// TIA Portal V17 export
// export: Created 2025-06-26T06:49:14.7827418Z, ExportSetting WithDefaults, DisplayName Totally Integrated Automation Portal, DisplayVersion V17 Update 8, DisplayName TIA Portal Openness, DisplayVersion V17 Update 8, DisplayName TIA Portal Version Control Interface, DisplayVersion V17, DisplayName STEP 7 Professional, DisplayVersion V17 Update 8, DisplayName STEP 7 Safety, DisplayVersion V17 Update 6, DisplayName WinCC Advanced, DisplayVersion V17 Update 8
FUNCTION_BLOCK "ApplicationCommunication"   // FB6, LAD
{ S7_Optimized_Access := 'TRUE' }
VERSION : 0.1
// Note some networks are in Ladder because the FBD equivalents are too bulky and the SCL equivalents are too easy to screw up accidentally.
// stored: AutoNumber true, IsIECCheckEnabled false, IsRetainMemResEnabled false, MemoryReserve 0, SetENOAutomatically false, UDAEnableTagReadback false
   VAR
      ExpansionRegulatorManualOn { ExternalAccessible := 'False'; ExternalVisible := 'False'; ExternalWritable := 'False'} : Bool;
      ExpansionRegulatorManualOff { ExternalAccessible := 'False'; ExternalVisible := 'False'; ExternalWritable := 'False'; S7_SetPoint := 'True'} : Bool;
      HeatSinkOutManualOn { ExternalAccessible := 'False'; ExternalVisible := 'False'; ExternalWritable := 'False'} : Bool;
      HeatSinkOutManualOff { ExternalAccessible := 'False'; ExternalVisible := 'False'; ExternalWritable := 'False'} : Bool;
      PerformanceManualModeOn { ExternalAccessible := 'False'; ExternalVisible := 'False'; ExternalWritable := 'False'} : Bool;
      PerformanceManualModeOff { ExternalAccessible := 'False'; ExternalVisible := 'False'; ExternalWritable := 'False'} : Bool;
      OilHeatingManualOn { ExternalAccessible := 'False'; ExternalVisible := 'False'; ExternalWritable := 'False'} : Bool;
      OilHeatingManualOff { ExternalAccessible := 'False'; ExternalVisible := 'False'; ExternalWritable := 'False'} : Bool;
      PinchManualModeOn { ExternalAccessible := 'False'; ExternalVisible := 'False'; ExternalWritable := 'False'} : Bool;
      PinchManualModeOff { ExternalAccessible := 'False'; ExternalVisible := 'False'; ExternalWritable := 'False'} : Bool;
      SuperheatManualOn { ExternalAccessible := 'False'; ExternalVisible := 'False'; ExternalWritable := 'False'} : Bool;
      SuperheatManualOff { ExternalAccessible := 'False'; ExternalVisible := 'False'; ExternalWritable := 'False'} : Bool;
      AlarmAckOn { ExternalAccessible := 'False'; ExternalVisible := 'False'; ExternalWritable := 'False'} : Bool;
      AlarmAckOff { ExternalAccessible := 'False'; ExternalVisible := 'False'; ExternalWritable := 'False'} : Bool;
      ResetEstopOn { ExternalAccessible := 'False'; ExternalVisible := 'False'; ExternalWritable := 'False'} : Bool;
      ResetEstopOff { ExternalAccessible := 'False'; ExternalVisible := 'False'; ExternalWritable := 'False'} : Bool;
      FastStopOn { ExternalAccessible := 'False'; ExternalVisible := 'False'; ExternalWritable := 'False'} : Bool;
      ExpansionManualPrev { ExternalAccessible := 'False'; ExternalVisible := 'False'; ExternalWritable := 'False'} : Real;
      HeatSinkManualPrev { ExternalAccessible := 'False'; ExternalVisible := 'False'; ExternalWritable := 'False'} : Real;
      PerformanceManualPrev { ExternalAccessible := 'False'; ExternalVisible := 'False'; ExternalWritable := 'False'} : Real;
      OilHeatingManualPrev { ExternalAccessible := 'False'; ExternalVisible := 'False'; ExternalWritable := 'False'} : Real;
      PinchManualPrev { ExternalAccessible := 'False'; ExternalVisible := 'False'; ExternalWritable := 'False'} : Real;
      SuperheatManualPrev { ExternalAccessible := 'False'; ExternalVisible := 'False'; ExternalWritable := 'False'} : Real;
      HeatboosterSetpointPrev { ExternalAccessible := 'False'; ExternalVisible := 'False'; ExternalWritable := 'False'} : Real;
      RegulationTargetPrev { ExternalAccessible := 'False'; ExternalVisible := 'False'; ExternalWritable := 'False'} : Int;
      S7Watchdog : "fbHeartbeatCount2";
   END_VAR
   VAR_TEMP
      bDummy : Bool;
      fDummy : Real;
   END_VAR
   VAR_TEMP   // added for the SCL form of the ladder/FBD networks
      _w1 : Bool;
      _w2 : Bool;
      _w3 : Bool;
      _w4 : Bool;
      _w5 : Bool;
      _w6 : Bool;
      _w7 : Bool;
      _w8 : Bool;
      _w9 : Bool;
      _w10 : Bool;
   END_VAR
BEGIN

REGION Network 1 (SCL): Status
   // Applications PLC GETs these.
   "DB_Application".FromHB.EmergencyStop       := "DB_System".bEmergencyStop;
   "DB_Application".FromHB.OilHeatersGroup1    := "DB_DO".HBL_EC_01;
   "DB_Application".FromHB.OilHeatersGroup2    := "DB_DO".HBL_EC_02;
   "DB_Application".FromHB.HBL_SC_10_Ready     := "DB_InverterDrives".HBL_SC_10.Stat.bReady;
   "DB_Application".FromHB.HBL_SC_10_Run       := "DB_InverterDrives".HBL_SC_10.Stat.bRun;
   "DB_Application".FromHB.HBL_HV_630           := "DB_DO".HBL_HV_630;
   "DB_Application".FromHB.CPC_P_01            := "DB_DO".CPC_P_01;
   "DB_Application".FromHB.SSC_P_01            := "DB_DO".SSC_P_01;
   "DB_Application".FromHB.HBL_SC_10_Tripped   := "DB_InverterDrives".HBL_SC_10.Stat.bTrip;
   "DB_Application".FromHB.HBL_SC_02_Ready     := "DB_InverterDrives".HBL_SC_02.Stat.bReady;
   "DB_Application".FromHB.HBL_SC_02_Run       := "DB_InverterDrives".HBL_SC_02.Stat.bRun;
   "DB_Application".FromHB.HBL_SC_02_Tripped   := "DB_InverterDrives".HBL_SC_02.Stat.bTrip;
   "DB_Application".FromHB.SSC_F_01            := "DB_DO".SSC_F_01;
   "DB_Application".FromHB.SSC_P_02            := "DB_DO".SSC_P_02;
   "DB_Application".FromHB.HBL_LS_01           := "DB_DI".HBL_LS_01.bValue;
   "DB_Application".FromHB.HBL_LS_02           := "DB_DI".HBL_LS_02.bValue;
   "DB_Application".FromHB.MachineState        := "DB_State".State.State_Number;
   "DB_Application".FromHB.CompressorType      := "DB_CurrentSetting".Compressor.CompressorTypeNumber;
   "DB_Application".FromHB.SystemType          := "DB_CurrentSetting".System.SystemTypeNumber;
   "DB_Application".FromHB.RefrigerantType     := "DB_CurrentSetting".Fluid.FluidTypeNumber;
   "DB_Application".FromHB.UptimeHours         := UDINT_TO_INT("DB_System".SystemUptime.nHours);
   "DB_Application".FromHB.UptimeMinutes       := "DB_System".SystemUptime.nMinutes;
   "DB_Application".FromHB.UptimeSeconds       := "DB_System".SystemUptime.nSeconds;
   "DB_Application".FromHB.ActiveTimeHours     := UDINT_TO_INT("DB_System".SystemActiveTime.nHours);
   "DB_Application".FromHB.ActiveTimeMinutes   := "DB_System".SystemActiveTime.nMinutes;
   "DB_Application".FromHB.ActiveTimeSeconds   := "DB_System".SystemActiveTime.nSeconds;
   "DB_Application".FromHB.RunningTimeHours    := UDINT_TO_INT("DB_System".RunningTime.nHours);
   "DB_Application".FromHB.RunningTimeMinutes  := "DB_System".RunningTime.nMinutes;
   "DB_Application".FromHB.RunningTimeSeconds  := "DB_System".RunningTime.nSeconds;
   "DB_Application".FromHB.HeatboosterSetpoint := "DB_Regulators".HeatboosterSetpoint;
   "DB_Application".FromHB.RegulationTarget    := "DB_Regulators".RegulationTarget;
   "DB_Application".FromHB.HBL_HCV_514_Force   := FALSE; // ###FIX
   "DB_Application".FromHB.HBL_HCV_514         := 5.14; //##FIX
   "DB_Application".FromHB.HBL_HCV_548_Force   := FALSE; // ##FIX
   "DB_Application".FromHB.HBL_HCV_548         := 5.48; //##FIX
END_REGION

REGION Network 2 (SCL): DB_AI
   // Copy only .fValues for minimum bandwidth
   "DB_Application".FromHB.DB_AI.HBL_TT_502 := "DB_AI".HBL_TT_502.Eng.fValue;
   "DB_Application".FromHB.DB_AI.HBL_PT_503 := "DB_AI".HBL_PT_503.Eng.fValue;
   "DB_Application".FromHB.DB_AI.HBL_TT_504 := "DB_AI".HBL_TT_504.Eng.fValue;
   "DB_Application".FromHB.DB_AI.HBL_LT_510 := "DB_AI".HBL_LT_510.Eng.fValue;
   "DB_Application".FromHB.DB_AI.HBL_PT_511 := "DB_AI".HBL_PT_511.Eng.fValue;
   "DB_Application".FromHB.DB_AI.HBL_TT_512 := "DB_AI".HBL_TT_512.Eng.fValue;
   "DB_Application".FromHB.DB_AI.HBL_TT_516 := "DB_AI".HBL_TT_516.Eng.fValue;
   "DB_Application".FromHB.DB_AI.HBL_PT_517 := "DB_AI".HBL_PT_517.Eng.fValue;
   "DB_Application".FromHB.DB_AI.HBL_TT_518 := "DB_AI".HBL_TT_518.Eng.fValue;
   "DB_Application".FromHB.DB_AI.HBL_PT_519 := "DB_AI".HBL_PT_519.Eng.fValue;
   "DB_Application".FromHB.DB_AI.HBL_FT_520 := "DB_AI".HBL_FT_520.Eng.fValue;
   "DB_Application".FromHB.DB_AI.HBL_TT_530 := "DB_AI".HBL_TT_530.Eng.fValue;
   "DB_Application".FromHB.DB_AI.HBL_PT_531 := "DB_AI".HBL_PT_531.Eng.fValue;
   "DB_Application".FromHB.DB_AI.HBL_TT_532 := "DB_AI".HBL_TT_532.Eng.fValue;
   "DB_Application".FromHB.DB_AI.HBL_TT_533 := "DB_AI".HBL_TT_533.Eng.fValue;
   "DB_Application".FromHB.DB_AI.HBL_PT_534 := "DB_AI".HBL_PT_534.Eng.fValue;
   "DB_Application".FromHB.DB_AI.HBL_AT_535 := "DB_AI".HBL_AT_535.Eng.fValue;
   "DB_Application".FromHB.DB_AI.HBL_TT_540 := "DB_AI".HBL_TT_540.Eng.fValue;
   "DB_Application".FromHB.DB_AI.HBL_PT_541 := "DB_AI".HBL_PT_541.Eng.fValue;
   "DB_Application".FromHB.DB_AI.HBL_TT_542 := "DB_AI".HBL_TT_542.Eng.fValue;
   "DB_Application".FromHB.DB_AI.HBL_TT_543 := "DB_AI".HBL_TT_543.Eng.fValue;
   "DB_Application".FromHB.DB_AI.HBL_PT_544 := "DB_AI".HBL_PT_544.Eng.fValue;
   "DB_Application".FromHB.DB_AI.HBL_AT_545 := "DB_AI".HBL_AT_545.Eng.fValue;
   "DB_Application".FromHB.DB_AI.HBL_TT_546 := "DB_AI".HBL_TT_546.Eng.fValue;
   "DB_Application".FromHB.DB_AI.HBL_PT_547 := "DB_AI".HBL_PT_547.Eng.fValue;
   "DB_Application".FromHB.DB_AI.HBL_TT_571 := "DB_AI".HBL_TT_571.Eng.fValue;
   "DB_Application".FromHB.DB_AI.HBL_PT_572 := "DB_AI".HBL_PT_572.Eng.fValue;
   "DB_Application".FromHB.DB_AI.HBL_TT_573 := "DB_AI".HBL_TT_573.Eng.fValue;
   "DB_Application".FromHB.DB_AI.HBL_LT_610 := "DB_AI".HBL_LT_610.Eng.fValue;
   "DB_Application".FromHB.DB_AI.HBL_TT_611 := "DB_AI".HBL_TT_611.Eng.fValue;
   "DB_Application".FromHB.DB_AI.HBL_PT_612 := "DB_AI".HBL_PT_612.Eng.fValue;
   "DB_Application".FromHB.DB_AI.HBL_CT_615 := "DB_AI".HBL_CT_615.Eng.fValue;
   "DB_Application".FromHB.DB_AI.HBL_PT_618 := "DB_AI".HBL_PT_618.Eng.fValue;
   "DB_Application".FromHB.DB_AI.HBL_PT_635 := "DB_AI".HBL_PT_635.Eng.fValue;
   "DB_Application".FromHB.DB_AI.HBL_PT_636 := "DB_AI".HBL_PT_636.Eng.fValue;
   "DB_Application".FromHB.DB_AI.HBL_LT_650 := "DB_AI".HBL_LT_650.Eng.fValue;
   "DB_Application".FromHB.DB_AI.HBL_PT_651 := "DB_AI".HBL_PT_651.Eng.fValue;
   "DB_Application".FromHB.DB_AI.HBL_PT_701 := "DB_AI".HBL_PT_701.Eng.fValue;
   "DB_Application".FromHB.DB_AI.HBL_PT_702 := "DB_AI".HBL_PT_702.Eng.fValue;
   "DB_Application".FromHB.DB_AI.HBL_PT_703 := "DB_AI".HBL_PT_703.Eng.fValue;

   "DB_Application".FromHB.DB_AI.CPC_LT_870 := "DB_AI".CPC_LT_870.Eng.fValue;
   "DB_Application".FromHB.DB_AI.CPC_TT_871 := "DB_AI".CPC_TT_871.Eng.fValue;
   "DB_Application".FromHB.DB_AI.CPC_PT_872 := "DB_AI".CPC_PT_872.Eng.fValue;
   "DB_Application".FromHB.DB_AI.CPC_PT_862 := "DB_AI".CPC_PT_862.Eng.fValue;
   "DB_Application".FromHB.DB_AI.HBL_TT_901 := "DB_AI".HBL_TT_901.Eng.fValue;
   "DB_Application".FromHB.DB_AI.HBL_PT_902 := "DB_AI".HBL_PT_902.Eng.fValue;

   "DB_Application".FromHB.DB_AI.HBL_TT_03 := "DB_AI".HBL_TT_03.Eng.fValue;
   "DB_Application".FromHB.DB_AI.HBL_TT_16 := "DB_AI".HBL_TT_16.Eng.fValue;
   "DB_Application".FromHB.DB_AI.HBL_TT_17 := "DB_AI".HBL_TT_17.Eng.fValue;
   "DB_Application".FromHB.DB_AI.HBL_TT_18 := "DB_AI".HBL_TT_18.Eng.fValue;
   "DB_Application".FromHB.DB_AI.HBL_TT_20 := "DB_AI".HBL_TT_20.Eng.fValue;
   "DB_Application".FromHB.DB_AI.HBL_TT_21 := "DB_AI".HBL_TT_21.Eng.fValue;
   "DB_Application".FromHB.DB_AI.HBL_TT_22 := "DB_AI".HBL_TT_22.Eng.fValue;
   "DB_Application".FromHB.DB_AI.HBL_TT_23 := "DB_AI".HBL_TT_23.Eng.fValue;
   "DB_Application".FromHB.DB_AI.HBL_TT_24 := "DB_AI".HBL_TT_24.Eng.fValue;
   "DB_Application".FromHB.DB_AI.HBL_TT_25 := "DB_AI".HBL_TT_25.Eng.fValue;
   "DB_Application".FromHB.DB_AI.HBL_TT_26 := "DB_AI".HBL_TT_26.Eng.fValue;
   "DB_Application".FromHB.DB_AI.HBL_TT_27 := "DB_AI".HBL_TT_27.Eng.fValue;
   "DB_Application".FromHB.DB_AI.HBL_PT_05 := "DB_AI".HBL_PT_05.Eng.fValue;
   "DB_Application".FromHB.DB_AI.HBL_PT_06 := "DB_AI".HBL_PT_960.Eng.fValue;
   "DB_Application".FromHB.DB_AI.HBL_PT_17 := "DB_AI".HBL_PT_961.Eng.fValue;
   "DB_Application".FromHB.DB_AI.HBL_CT_01 := "DB_AI".HBL_CT_01.Eng.fValue;
   "DB_Application".FromHB.DB_AI.HBL_CT_03 := "DB_AI".HBL_CT_950.Eng.fValue;

   "DB_Application".FromHB.DB_AI.SSC_TT_01 := "DB_AI".SSC_TT_01.Eng.fValue;
   "DB_Application".FromHB.DB_AI.SSC_TT_02 := "DB_AI".SSC_TT_02.Eng.fValue;
   "DB_Application".FromHB.DB_AI.SSC_TT_03 := "DB_AI".SSC_TT_03.Eng.fValue;
   "DB_Application".FromHB.DB_AI.SSC_TT_04 := "DB_AI".SSC_TT_04.Eng.fValue;
   "DB_Application".FromHB.DB_AI.SSC_PIT_01 := "DB_AI".SSC_PIT_01.Eng.fValue;
   "DB_Application".FromHB.DB_AI.SSC_PDT_01 := "DB_AI".SSC_PDT_01.Eng.fValue;
   "DB_Application".FromHB.DB_AI.SSC_LT_01 := "DB_AI".SSC_LT_01.Eng.fValue;
END_REGION

REGION Network 3 (SCL): DB_Calc
   // Done this way for minimum bandwidth
   "DB_Application".FromHB.DB_Calc.Compressor_CrankcaseSaturationTemperature   := "DB_Calc".Compressor.CrankcaseSaturationTemperature.fValue;
   "DB_Application".FromHB.DB_Calc.Compressor_CrankcaseSuperheat               := "DB_Calc".Compressor.CrankcaseSuperheat.fValue;
   "DB_Application".FromHB.DB_Calc.Compressor_VolumetricEfficiency             := "DB_Calc".Compressor.VolumetricEfficiency.fValue;
   "DB_Application".FromHB.DB_Calc.Compressor_IsentropicEfficiency             := "DB_Calc".Compressor.IsentropicEfficiency.fValue;
   "DB_Application".FromHB.DB_Calc.Compressor_Massflow                         := "DB_Calc".Compressor.Massflow.fValue;

   "DB_Application".FromHB.DB_Calc.Heatsink_DeltaT                             := "DB_Calc".HeatSink.DeltaT.fValue;
   "DB_Application".FromHB.DB_Calc.Heatsink_Pinch                              := "DB_Calc".HeatSink.Pinch.fValue;
   "DB_Application".FromHB.DB_Calc.Heatsink_Heatrate                           := "DB_Calc".HeatSink.HeatRate.fValue;
   "DB_Application".FromHB.DB_Calc.Heatsink_DeltaP                             := "DB_Calc".HeatSink.DeltaP.fValue;
   "DB_Application".FromHB.DB_Calc.Heatsink_Massflow                           := "DB_Calc".HeatSink.Massflow.fValue;

   "DB_Application".FromHB.DB_Calc.Heatsource_DeltaT                           := "DB_Calc".HeatSource.DeltaT.fValue;
   "DB_Application".FromHB.DB_Calc.Heatsource_Pinch                            := "DB_Calc".HeatSource.Pinch.fValue;
   "DB_Application".FromHB.DB_Calc.Heatsource_Heatrate                         := "DB_Calc".HeatSource.HeatRate.fValue;
   "DB_Application".FromHB.DB_Calc.Heatsource_DeltaP                           := "DB_Calc".HeatSource.DeltaP.fValue;
   "DB_Application".FromHB.DB_Calc.Heatsource_Massflow                         := "DB_Calc".HeatSource.Massflow.fValue;
   "DB_Application".FromHB.DB_Calc.Heatsource_TemperatureRateOfChange          := "DB_Calc".HeatSource.TemperatureRateOfChange.fValue;

   "DB_Application".FromHB.DB_Calc.HighPressPart_CompressorSaturationTemperature := "DB_Calc".HighPressPart.CompressorSaturationTemperature.fValue;
   "DB_Application".FromHB.DB_Calc.HighPressPart_CompressorSuperheat           := "DB_Calc".HighPressPart.CompressorSuperheat.fValue;
   "DB_Application".FromHB.DB_Calc.HighPressPart_CondenserSaturationTemperature:= "DB_Calc".HighPressPart.CondenserSaturationTemperature.fValue;
   "DB_Application".FromHB.DB_Calc.HighPressPart_CondenserSubcooling           := "DB_Calc".HighPressPart.CondenserSubcooling.fValue;
   "DB_Application".FromHB.DB_Calc.HighPressPart_ExpansionValveSubcooling      := "DB_Calc".HighPressPart.ExpansionValveSubcooling.fValue;
   "DB_Application".FromHB.DB_Calc.HighPressPart_CondenserDeltaP               := "DB_Calc".HighPressPart.CondenserDeltaP.fValue;

   "DB_Application".FromHB.DB_Calc.LowPressPart_EvaporatorSuperheat            := "DB_Calc".LowPressPart.EvaporatorSuperheat.fValue;
   "DB_Application".FromHB.DB_Calc.LowPressPart_CompressorSuperheat            := "DB_Calc".LowPressPart.CompressorSuperheat.fValue;
   "DB_Application".FromHB.DB_Calc.LowPressPart_EvaporatorSaturationTemperature:= "DB_Calc".LowPressPart.EvaporatorSaturationTemperature.fValue;
   "DB_Application".FromHB.DB_Calc.LowPressPart_CompressorSaturationTemperature:= "DB_Calc".LowPressPart.CompressorSaturationTemperature.fValue;

   "DB_Application".FromHB.DB_Calc.System_Quality                              := "DB_Calc".System.Quality.fValue;
   "DB_Application".FromHB.DB_Calc.System_COP                                  := "DB_Calc".System.COP.fValue;
   "DB_Application".FromHB.DB_Calc.System_ElectricalPower                      := "DB_Calc".System.ElectricalPower.fValue;
   "DB_Application".FromHB.DB_Calc.System_TemperatureLift                      := "DB_Calc".System.TemperatureLift.fValue;
   "DB_Application".FromHB.DB_Calc.System_MotorEfficiency                      := "DB_Calc".System.MotorEfficiency.fValue;
   "DB_Application".FromHB.DB_Calc.System_FMEP                                 := "DB_Calc".System.FMEP.fValue;

   "DB_Application".FromHB.DB_Calc.Aux_ShaftSealDeltaT                         := "DB_Calc".Auxiliary.ShaftSealDeltaT.fValue;
   "DB_Application".FromHB.DB_Calc.Aux_CPCPumpDeltaP                           := "DB_Calc".Auxiliary.CPCDeltaP.fValue;

   "DB_Application".FromHB.DB_Calc.Misc_EvaporatorDischargePressureMean        := "DB_Calc".Misc.EvaporatorDischargePressureMean.fValue;
   "DB_Application".FromHB.DB_Calc.Misc_EvaporatorDischargeTemperatureMin      := "DB_Calc".Misc.EvaporatorDischargeTemperatureMin.fValue;
   "DB_Application".FromHB.DB_Calc.Misc_EvaporatorDischargeTemperatureMean     := "DB_Calc".Misc.EvaporatorDischargeTemperatureMean.fValue;
   "DB_Application".FromHB.DB_Calc.Misc_OilFilterDeltaP                        := "DB_Calc".Misc.OilFilterDeltaP.fValue;
END_REGION

REGION Network 4 (SCL): DB_InverterDrives & DB_Valves
   // Done this way for minimum bandwidth
   "DB_Application".FromHB.DB_InverterDrives.HBL_SC_01_A1  := "DB_InverterDrives".HBL_SC_01.Stat.Speed.Eng.fValue;
   "DB_Application".FromHB.DB_InverterDrives.HBL_SC_01_A2  := "DB_InverterDrives".HBL_SC_01.Stat.Torque.Eng.fValue;
   "DB_Application".FromHB.DB_InverterDrives.HBL_SC_01_A3  := "DB_InverterDrives".HBL_SC_01.Stat.Power.Eng.fValue;
   "DB_Application".FromHB.DB_InverterDrives.HBL_SC_02_A1  := "DB_InverterDrives".HBL_SC_02.Stat.Speed.Eng.fValue;
   "DB_Application".FromHB.DB_InverterDrives.HBL_SC_02_A2  := "DB_InverterDrives".HBL_SC_02.Stat.Torque.Eng.fValue;
   "DB_Application".FromHB.DB_InverterDrives.HBL_SC_02_A3  := "DB_InverterDrives".HBL_SC_02.Stat.Power.Eng.fValue;
   "DB_Application".FromHB.DB_InverterDrives.HBL_SC_10_A1  := "DB_InverterDrives".HBL_SC_10.Stat.Speed.Eng.fValue;
   "DB_Application".FromHB.DB_InverterDrives.HBL_SC_10_A2  := "DB_InverterDrives".HBL_SC_10.Stat.Torque.Eng.fValue;
   "DB_Application".FromHB.DB_InverterDrives.HBL_SC_10_A3  := "DB_InverterDrives".HBL_SC_10.Stat.Power.Eng.fValue;
   "DB_Application".FromHB.DB_InverterDrives.HBL_SC_03_A1  := "DB_InverterDrives".HBL_SC_03.Stat.Speed.Eng.fValue;
   "DB_Application".FromHB.DB_InverterDrives.HBL_SC_03_A2  := "DB_InverterDrives".HBL_SC_03.Stat.Torque.Eng.fValue;
   "DB_Application".FromHB.DB_InverterDrives.HBL_SC_03_A3  := "DB_InverterDrives".HBL_SC_03.Stat.Power.Eng.fValue;

   "DB_Application".FromHB.DB_Valves.HBL_HCV_576_A1        := "DB_Valves".HBL_HCV_576.Stat.Position.Eng.fValue;
   "DB_Application".FromHB.DB_Valves.HBL_HCV_577_A1        := "DB_Valves".HBL_HCV_577.Stat.Position.Eng.fValue;
   "DB_Application".FromHB.DB_Valves.HBL_HCV_578_A1        := "DB_Valves".HBL_HCV_578.Stat.Position.Eng.fValue;
   "DB_Application".FromHB.DB_Valves.HBL_HCV_579_A1        := "DB_Valves".HBL_HCV_579.Stat.Position.Eng.fValue;
   "DB_Application".FromHB.DB_Valves.HBL_HCV_515_A1        := "DB_Valves".HBL_HCV_515.Stat.Position.Eng.fValue;
   "DB_Application".FromHB.DB_Valves.HBL_HCV_575_A1        := "DB_Valves".HBL_HCV_575.Stat.Position.Eng.fValue;
   "DB_Application".FromHB.DB_Valves.HBL_HCV_616_A1        := "DB_Valves".HBL_HCV_616.Stat.Position.Eng.fValue;
   "DB_Application".FromHB.DB_Valves.HBL_HCV_700_A1        := "DB_Valves".HBL_HCV_700.Stat.Position.Eng.fValue;
   "DB_Application".FromHB.DB_Valves.HBL_HCV_514_A1        := "DB_Valves".HBL_HCV_514.Stat.Position.Eng.fValue;
   "DB_Application".FromHB.DB_Valves.HBL_HCV_548_A1        := "DB_Valves".HBL_HCV_548.Stat.Position.Eng.fValue;
END_REGION

REGION Network 5 (SCL): Commands
   // Application PLC PUTs these, so no code here :-)
END_REGION

REGION Network 6: Watchdog/liveness bit
   // Check if data is valid from external systems
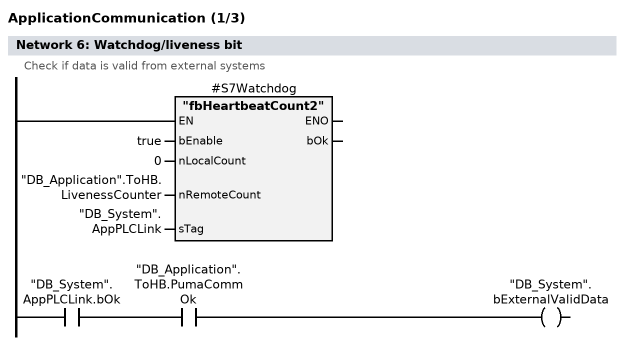
   RUNG wire#powerrail
      #S7Watchdog(bEnable := true, nLocalCount := 0, nRemoteCount := "DB_Application".ToHB.LivenessCounter, sTag := "DB_System".AppPLCLink, bOk =>)
   END_RUNG
   RUNG wire#powerrail
      Contact( "DB_System".AppPLCLink.bOk )
      Contact( "DB_Application".ToHB.PumaCommOk )
      Coil( "DB_System".bExternalValidData )
   END_RUNG
   // the same network as SCL:
   #S7Watchdog(bEnable := true,   // "fbHeartbeatCount2"
               nLocalCount := 0,
               nRemoteCount := "DB_Application".ToHB.LivenessCounter,
               sTag := "DB_System".AppPLCLink);
   "DB_System".bExternalValidData := "DB_System".AppPLCLink.bOk AND "DB_Application".ToHB.PumaCommOk;
END_REGION

REGION Network 7: Process setpoints from Application PLC
   // A positive edge followed by a SET  writes to the destination bit once, without "holding" the value. Easiest to write & read in ladder.
   // Triggering a MOVE on value change writes the value once without continually overwriting it.
   // A negative edge followed by a RESET writes to the destination bit once, without "holding" the value. Easiest to write & read in ladder.
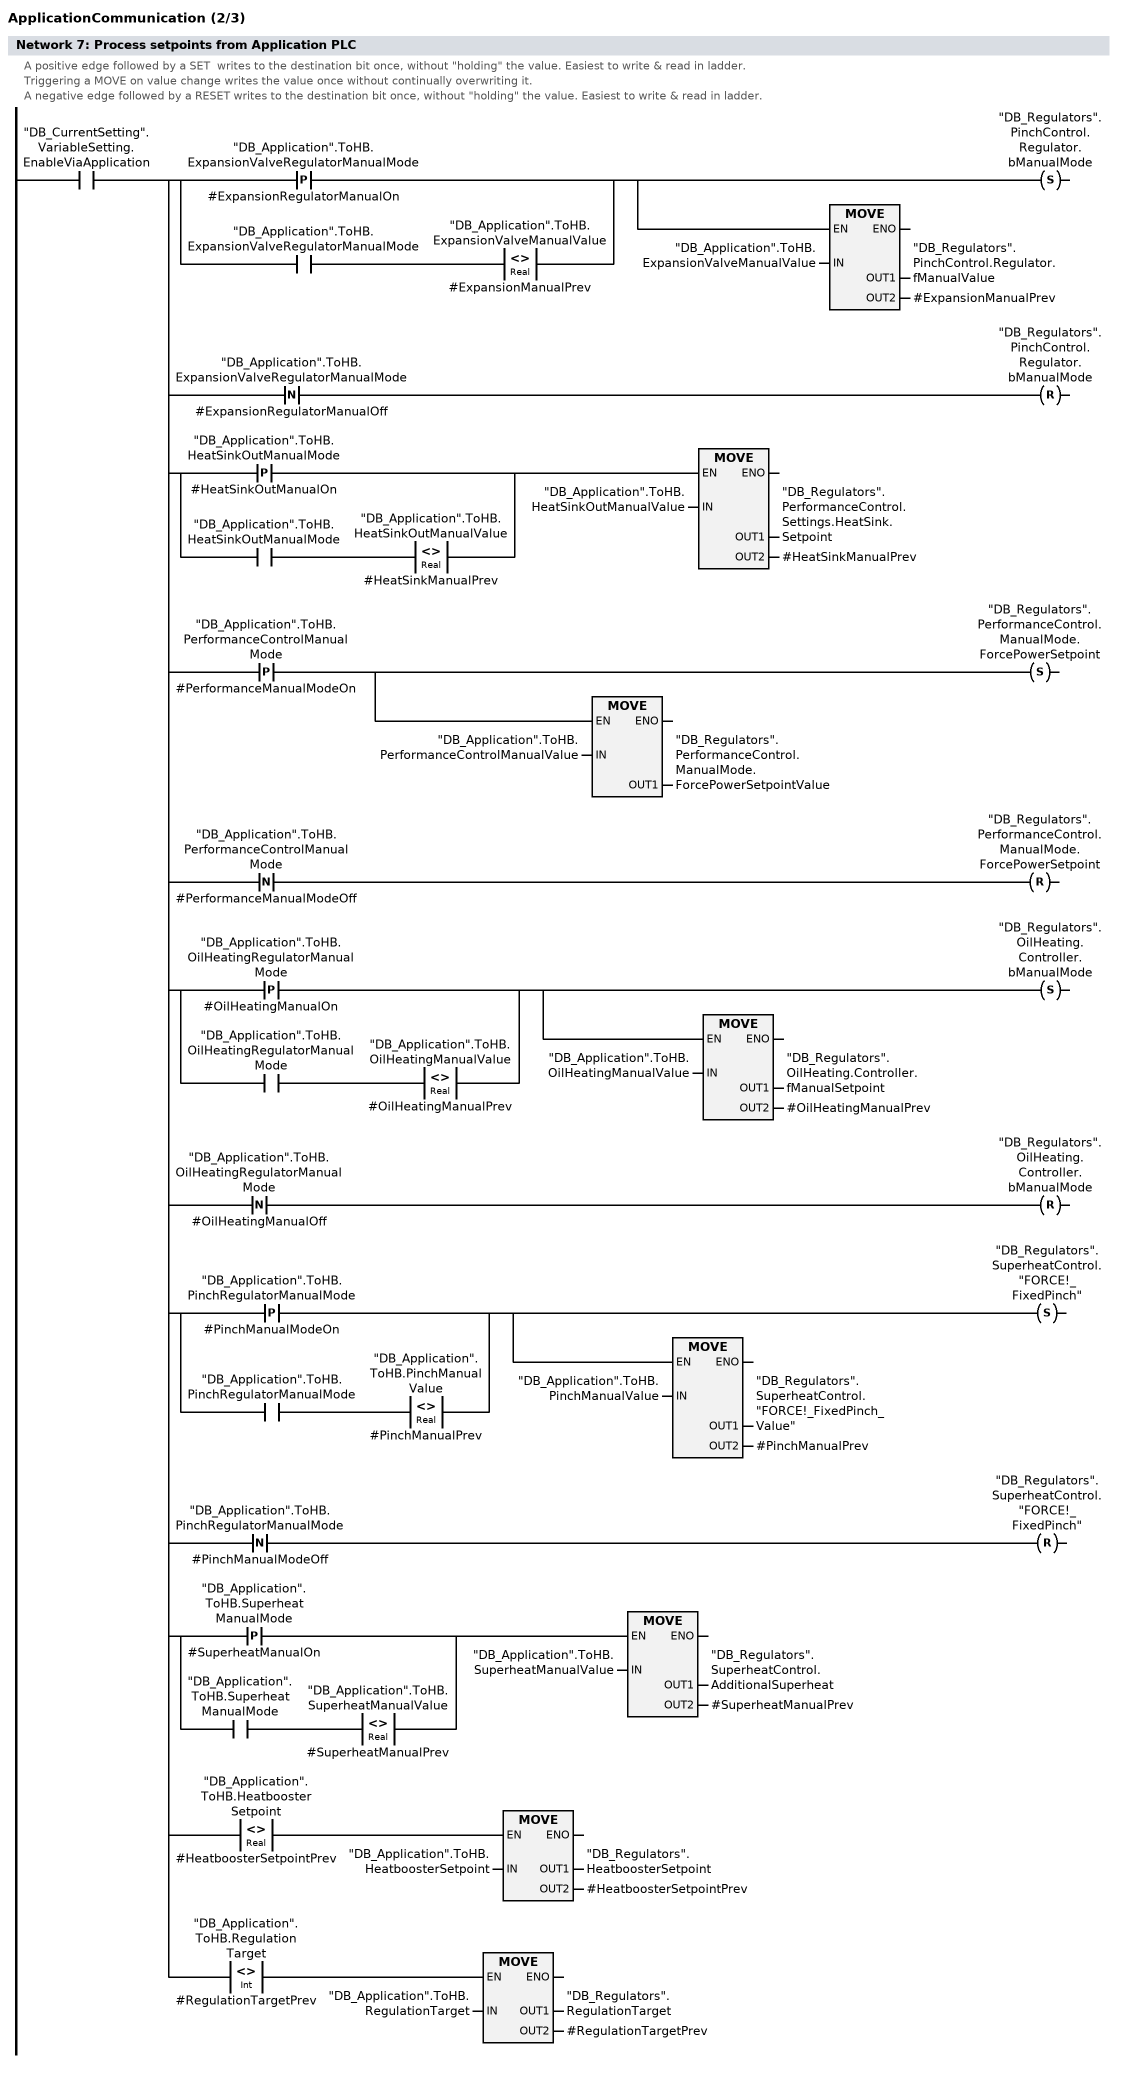
   RUNG wire#powerrail
      Contact( "DB_CurrentSetting".VariableSetting.EnableViaApplication )
      wire#w1
      P_Contact(operand := "DB_Application".ToHB.ExpansionValveRegulatorManualMode, bit := #ExpansionRegulatorManualOn)
      wire#w2
      S_Coil( "DB_Regulators".PinchControl.Regulator.bManualMode )
   END_RUNG
   RUNG wire#w1
      Contact( "DB_Application".ToHB.ExpansionValveRegulatorManualMode )
      { S7_Templates := "SrcType := Real" } NE_Contact(in1 := "DB_Application".ToHB.ExpansionValveManualValue, in2 := #ExpansionManualPrev)
   END_RUNG wire#w2
   RUNG wire#w2
      Move(in := "DB_Application".ToHB.ExpansionValveManualValue, out1 => "DB_Regulators".PinchControl.Regulator.fManualValue, out2 => #ExpansionManualPrev)
   END_RUNG
   RUNG wire#w1
      N_Contact(operand := "DB_Application".ToHB.ExpansionValveRegulatorManualMode, bit := #ExpansionRegulatorManualOff)
      R_Coil( "DB_Regulators".PinchControl.Regulator.bManualMode )
   END_RUNG
   RUNG wire#w1
      P_Contact(operand := "DB_Application".ToHB.HeatSinkOutManualMode, bit := #HeatSinkOutManualOn)
      wire#w3
      Move(in := "DB_Application".ToHB.HeatSinkOutManualValue, out1 => "DB_Regulators".PerformanceControl.Settings.HeatSink.Setpoint, out2 => #HeatSinkManualPrev)
   END_RUNG
   RUNG wire#w1
      Contact( "DB_Application".ToHB.HeatSinkOutManualMode )
      { S7_Templates := "SrcType := Real" } NE_Contact(in1 := "DB_Application".ToHB.HeatSinkOutManualValue, in2 := #HeatSinkManualPrev)
   END_RUNG wire#w3
   RUNG wire#w1
      P_Contact(operand := "DB_Application".ToHB.PerformanceControlManualMode, bit := #PerformanceManualModeOn)
      wire#w4
      S_Coil( "DB_Regulators".PerformanceControl.ManualMode.ForcePowerSetpoint )
   END_RUNG
   RUNG wire#w4
      Move(in := "DB_Application".ToHB.PerformanceControlManualValue, out1 => "DB_Regulators".PerformanceControl.ManualMode.ForcePowerSetpointValue)
   END_RUNG
   RUNG wire#w1
      N_Contact(operand := "DB_Application".ToHB.PerformanceControlManualMode, bit := #PerformanceManualModeOff)
      R_Coil( "DB_Regulators".PerformanceControl.ManualMode.ForcePowerSetpoint )
   END_RUNG
   RUNG wire#w1
      P_Contact(operand := "DB_Application".ToHB.OilHeatingRegulatorManualMode, bit := #OilHeatingManualOn)
      wire#w5
      S_Coil( "DB_Regulators".OilHeating.Controller.bManualMode )
   END_RUNG
   RUNG wire#w1
      Contact( "DB_Application".ToHB.OilHeatingRegulatorManualMode )
      { S7_Templates := "SrcType := Real" } NE_Contact(in1 := "DB_Application".ToHB.OilHeatingManualValue, in2 := #OilHeatingManualPrev)
   END_RUNG wire#w5
   RUNG wire#w5
      Move(in := "DB_Application".ToHB.OilHeatingManualValue, out1 => "DB_Regulators".OilHeating.Controller.fManualSetpoint, out2 => #OilHeatingManualPrev)
   END_RUNG
   RUNG wire#w1
      N_Contact(operand := "DB_Application".ToHB.OilHeatingRegulatorManualMode, bit := #OilHeatingManualOff)
      R_Coil( "DB_Regulators".OilHeating.Controller.bManualMode )
   END_RUNG
   RUNG wire#w1
      P_Contact(operand := "DB_Application".ToHB.PinchRegulatorManualMode, bit := #PinchManualModeOn)
      wire#w6
      S_Coil( "DB_Regulators".SuperheatControl."FORCE!_FixedPinch" )
   END_RUNG
   RUNG wire#w1
      Contact( "DB_Application".ToHB.PinchRegulatorManualMode )
      { S7_Templates := "SrcType := Real" } NE_Contact(in1 := "DB_Application".ToHB.PinchManualValue, in2 := #PinchManualPrev)
   END_RUNG wire#w6
   RUNG wire#w6
      Move(in := "DB_Application".ToHB.PinchManualValue, out1 => "DB_Regulators".SuperheatControl."FORCE!_FixedPinch_Value", out2 => #PinchManualPrev)
   END_RUNG
   RUNG wire#w1
      N_Contact(operand := "DB_Application".ToHB.PinchRegulatorManualMode, bit := #PinchManualModeOff)
      R_Coil( "DB_Regulators".SuperheatControl."FORCE!_FixedPinch" )
   END_RUNG
   RUNG wire#w1
      P_Contact(operand := "DB_Application".ToHB.SuperheatManualMode, bit := #SuperheatManualOn)
      wire#w7
      Move(in := "DB_Application".ToHB.SuperheatManualValue, out1 => "DB_Regulators".SuperheatControl.AdditionalSuperheat, out2 => #SuperheatManualPrev)
   END_RUNG
   RUNG wire#w1
      Contact( "DB_Application".ToHB.SuperheatManualMode )
      { S7_Templates := "SrcType := Real" } NE_Contact(in1 := "DB_Application".ToHB.SuperheatManualValue, in2 := #SuperheatManualPrev)
   END_RUNG wire#w7
   RUNG wire#w1
      { S7_Templates := "SrcType := Real" } NE_Contact(in1 := "DB_Application".ToHB.HeatboosterSetpoint, in2 := #HeatboosterSetpointPrev)
      Move(in := "DB_Application".ToHB.HeatboosterSetpoint, out1 => "DB_Regulators".HeatboosterSetpoint, out2 => #HeatboosterSetpointPrev)
   END_RUNG
   RUNG wire#w1
      { S7_Templates := "SrcType := Int" } NE_Contact(in1 := "DB_Application".ToHB.RegulationTarget, in2 := #RegulationTargetPrev)
      Move(in := "DB_Application".ToHB.RegulationTarget, out1 => "DB_Regulators".RegulationTarget, out2 => #RegulationTargetPrev)
   END_RUNG
   // the same network as SCL:
   #_w1 := "DB_CurrentSetting".VariableSetting.EnableViaApplication AND "DB_Application".ToHB.ExpansionValveRegulatorManualMode AND NOT #ExpansionRegulatorManualOn;   // rising edge of "DB_Application".ToHB.ExpansionValveRegulatorManualMode
   #ExpansionRegulatorManualOn := "DB_Application".ToHB.ExpansionValveRegulatorManualMode;
   IF #_w1 OR ("DB_CurrentSetting".VariableSetting.EnableViaApplication AND "DB_Application".ToHB.ExpansionValveRegulatorManualMode AND ("DB_Application".ToHB.ExpansionValveManualValue <> #ExpansionManualPrev)) THEN
       "DB_Regulators".PinchControl.Regulator.bManualMode := TRUE;
       "DB_Regulators".PinchControl.Regulator.fManualValue := "DB_Application".ToHB.ExpansionValveManualValue;
       #ExpansionManualPrev := "DB_Application".ToHB.ExpansionValveManualValue;
   END_IF;
   #_w2 := "DB_CurrentSetting".VariableSetting.EnableViaApplication AND NOT "DB_Application".ToHB.ExpansionValveRegulatorManualMode AND #ExpansionRegulatorManualOff;   // falling edge of "DB_Application".ToHB.ExpansionValveRegulatorManualMode
   #ExpansionRegulatorManualOff := "DB_Application".ToHB.ExpansionValveRegulatorManualMode;
   IF #_w2 THEN "DB_Regulators".PinchControl.Regulator.bManualMode := FALSE; END_IF;
   #_w3 := "DB_CurrentSetting".VariableSetting.EnableViaApplication AND "DB_Application".ToHB.HeatSinkOutManualMode AND NOT #HeatSinkOutManualOn;   // rising edge of "DB_Application".ToHB.HeatSinkOutManualMode
   #HeatSinkOutManualOn := "DB_Application".ToHB.HeatSinkOutManualMode;
   IF #_w3 OR ("DB_CurrentSetting".VariableSetting.EnableViaApplication AND "DB_Application".ToHB.HeatSinkOutManualMode AND ("DB_Application".ToHB.HeatSinkOutManualValue <> #HeatSinkManualPrev)) THEN
       "DB_Regulators".PerformanceControl.Settings.HeatSink.Setpoint := "DB_Application".ToHB.HeatSinkOutManualValue;
       #HeatSinkManualPrev := "DB_Application".ToHB.HeatSinkOutManualValue;
   END_IF;
   #_w4 := "DB_CurrentSetting".VariableSetting.EnableViaApplication AND "DB_Application".ToHB.PerformanceControlManualMode AND NOT #PerformanceManualModeOn;   // rising edge of "DB_Application".ToHB.PerformanceControlManualMode
   #PerformanceManualModeOn := "DB_Application".ToHB.PerformanceControlManualMode;
   IF #_w4 THEN
       "DB_Regulators".PerformanceControl.ManualMode.ForcePowerSetpoint := TRUE;
       "DB_Regulators".PerformanceControl.ManualMode.ForcePowerSetpointValue := "DB_Application".ToHB.PerformanceControlManualValue;
   END_IF;
   #_w5 := "DB_CurrentSetting".VariableSetting.EnableViaApplication AND NOT "DB_Application".ToHB.PerformanceControlManualMode AND #PerformanceManualModeOff;   // falling edge of "DB_Application".ToHB.PerformanceControlManualMode
   #PerformanceManualModeOff := "DB_Application".ToHB.PerformanceControlManualMode;
   IF #_w5 THEN "DB_Regulators".PerformanceControl.ManualMode.ForcePowerSetpoint := FALSE; END_IF;
   #_w6 := "DB_CurrentSetting".VariableSetting.EnableViaApplication AND "DB_Application".ToHB.OilHeatingRegulatorManualMode AND NOT #OilHeatingManualOn;   // rising edge of "DB_Application".ToHB.OilHeatingRegulatorManualMode
   #OilHeatingManualOn := "DB_Application".ToHB.OilHeatingRegulatorManualMode;
   IF #_w6 OR ("DB_CurrentSetting".VariableSetting.EnableViaApplication AND "DB_Application".ToHB.OilHeatingRegulatorManualMode AND ("DB_Application".ToHB.OilHeatingManualValue <> #OilHeatingManualPrev)) THEN
       "DB_Regulators".OilHeating.Controller.bManualMode := TRUE;
       "DB_Regulators".OilHeating.Controller.fManualSetpoint := "DB_Application".ToHB.OilHeatingManualValue;
       #OilHeatingManualPrev := "DB_Application".ToHB.OilHeatingManualValue;
   END_IF;
   #_w7 := "DB_CurrentSetting".VariableSetting.EnableViaApplication AND NOT "DB_Application".ToHB.OilHeatingRegulatorManualMode AND #OilHeatingManualOff;   // falling edge of "DB_Application".ToHB.OilHeatingRegulatorManualMode
   #OilHeatingManualOff := "DB_Application".ToHB.OilHeatingRegulatorManualMode;
   IF #_w7 THEN "DB_Regulators".OilHeating.Controller.bManualMode := FALSE; END_IF;
   #_w8 := "DB_CurrentSetting".VariableSetting.EnableViaApplication AND "DB_Application".ToHB.PinchRegulatorManualMode AND NOT #PinchManualModeOn;   // rising edge of "DB_Application".ToHB.PinchRegulatorManualMode
   #PinchManualModeOn := "DB_Application".ToHB.PinchRegulatorManualMode;
   IF #_w8 OR ("DB_CurrentSetting".VariableSetting.EnableViaApplication AND "DB_Application".ToHB.PinchRegulatorManualMode AND ("DB_Application".ToHB.PinchManualValue <> #PinchManualPrev)) THEN
       "DB_Regulators".SuperheatControl."FORCE!_FixedPinch" := TRUE;
       "DB_Regulators".SuperheatControl."FORCE!_FixedPinch_Value" := "DB_Application".ToHB.PinchManualValue;
       #PinchManualPrev := "DB_Application".ToHB.PinchManualValue;
   END_IF;
   #_w9 := "DB_CurrentSetting".VariableSetting.EnableViaApplication AND NOT "DB_Application".ToHB.PinchRegulatorManualMode AND #PinchManualModeOff;   // falling edge of "DB_Application".ToHB.PinchRegulatorManualMode
   #PinchManualModeOff := "DB_Application".ToHB.PinchRegulatorManualMode;
   IF #_w9 THEN "DB_Regulators".SuperheatControl."FORCE!_FixedPinch" := FALSE; END_IF;
   #_w10 := "DB_CurrentSetting".VariableSetting.EnableViaApplication AND "DB_Application".ToHB.SuperheatManualMode AND NOT #SuperheatManualOn;   // rising edge of "DB_Application".ToHB.SuperheatManualMode
   #SuperheatManualOn := "DB_Application".ToHB.SuperheatManualMode;
   IF #_w10 OR ("DB_CurrentSetting".VariableSetting.EnableViaApplication AND "DB_Application".ToHB.SuperheatManualMode AND ("DB_Application".ToHB.SuperheatManualValue <> #SuperheatManualPrev)) THEN
       "DB_Regulators".SuperheatControl.AdditionalSuperheat := "DB_Application".ToHB.SuperheatManualValue;
       #SuperheatManualPrev := "DB_Application".ToHB.SuperheatManualValue;
   END_IF;
   IF "DB_CurrentSetting".VariableSetting.EnableViaApplication AND ("DB_Application".ToHB.HeatboosterSetpoint <> #HeatboosterSetpointPrev) THEN
       "DB_Regulators".HeatboosterSetpoint := "DB_Application".ToHB.HeatboosterSetpoint;
       #HeatboosterSetpointPrev := "DB_Application".ToHB.HeatboosterSetpoint;
   END_IF;
   IF "DB_CurrentSetting".VariableSetting.EnableViaApplication AND ("DB_Application".ToHB.RegulationTarget <> #RegulationTargetPrev) THEN
       "DB_Regulators".RegulationTarget := "DB_Application".ToHB.RegulationTarget;
       #RegulationTargetPrev := "DB_Application".ToHB.RegulationTarget;
   END_IF;
END_REGION

REGION Network 8: Process commands from Application PLC
   // Start & stop requests handled by FB30 StartStopControl
   // FastStop handled by FB34 MotorControl
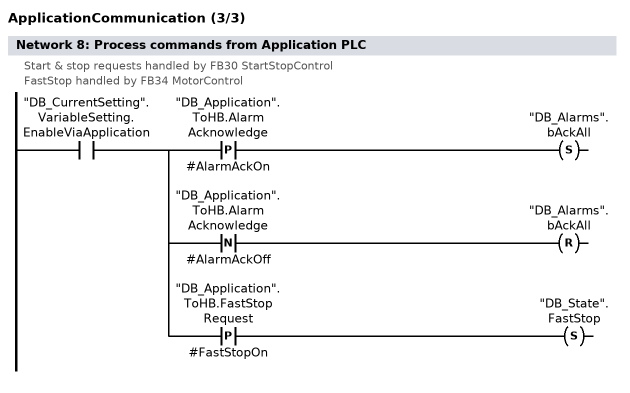
   RUNG wire#powerrail
      Contact( "DB_CurrentSetting".VariableSetting.EnableViaApplication )
      wire#w1
      P_Contact(operand := "DB_Application".ToHB.AlarmAcknowledge, bit := #AlarmAckOn)
      S_Coil( "DB_Alarms".bAckAll )
   END_RUNG
   RUNG wire#w1
      N_Contact(operand := "DB_Application".ToHB.AlarmAcknowledge, bit := #AlarmAckOff)
      R_Coil( "DB_Alarms".bAckAll )
   END_RUNG
   RUNG wire#w1
      P_Contact(operand := "DB_Application".ToHB.FastStopRequest, bit := #FastStopOn)
      S_Coil( "DB_State".FastStop )
   END_RUNG
   // the same network as SCL:
   #_w1 := "DB_CurrentSetting".VariableSetting.EnableViaApplication AND "DB_Application".ToHB.AlarmAcknowledge AND NOT #AlarmAckOn;   // rising edge of "DB_Application".ToHB.AlarmAcknowledge
   #AlarmAckOn := "DB_Application".ToHB.AlarmAcknowledge;
   IF #_w1 THEN "DB_Alarms".bAckAll := TRUE; END_IF;
   #_w2 := "DB_CurrentSetting".VariableSetting.EnableViaApplication AND NOT "DB_Application".ToHB.AlarmAcknowledge AND #AlarmAckOff;   // falling edge of "DB_Application".ToHB.AlarmAcknowledge
   #AlarmAckOff := "DB_Application".ToHB.AlarmAcknowledge;
   IF #_w2 THEN "DB_Alarms".bAckAll := FALSE; END_IF;
   #_w3 := "DB_CurrentSetting".VariableSetting.EnableViaApplication AND "DB_Application".ToHB.FastStopRequest AND NOT #FastStopOn;   // rising edge of "DB_Application".ToHB.FastStopRequest
   #FastStopOn := "DB_Application".ToHB.FastStopRequest;
   IF #_w3 THEN "DB_State".FastStop := TRUE; END_IF;
END_REGION
END_FUNCTION_BLOCK
